PROGRAM MAIN
VAR
	gGreenlight : BOOL := FALSE;
	yYellowlight : BOOL := FALSE;
	rRedLight : BOOL := FALSE;
	gGreenlighttimer : TON;
	yYellowlighttimer : TON;
	rRedlighttimer : TON;
END_VAR

gGreenlighttimer(IN := NOT rRedlighttimer.Q, PT := T#5S);

yYellowlighttimer(IN := gGreenlighttimer.Q, PT := T#2S);

rRedlighttimer(IN := yYellowlighttimer.Q, PT := T#5S);

gGreenlight := NOT gGreenlighttimer.Q AND gGreenlighttimer.IN;

yYellowlight := NOT yYellowlighttimer.Q AND yYellowlighttimer.IN;

rRedLight := NOT rRedlighttimer.Q AND rRedlighttimer.IN;

END_PROGRAM

(* stored: Version 1.1.0.1, ProductVersion 3.1.4024.16
   POU MAIN: Id {06295a7d-5590-4515-9abd-727d4b72425e}, SpecialFunc None *)
